FUNCTION_BLOCK CROSSCOMM_PEER_870DEA938BB7E735 (* Service Interface Function Block Type *)
  (* Standard: 61499-2 *)
  (* Version 0.0, 9/22/2017, bababen, nxtControl GmbH, template *)
  PACKAGE Main;
  (* Compiler Cpp nxtControl builtin 1.0 *)
  {SET_ATTRIBUTE(Runtime.FBType.ImplementingType, Runtime.System#DYNGEN_CROSSCOMM_PEER)}
  {SET_ATTRIBUTE(Configuration.GenericFBType.InterfaceParams, Runtime.System#<InterfaceList> <EventOutputs> <Event Name="INITO"> <With Var="ExtendPusher" /> </Event> <Event Name="CNF"> <With Var="ExtendPusher" /> </Event> </EventOutputs> <OutputVars> <VarDeclaration Name="ExtendPusher" Type="BOOL" /> </OutputVars> </InterfaceList>)}
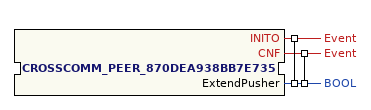
  EVENT_OUTPUT
    INITO WITH ExtendPusher;
    CNF WITH ExtendPusher;
  END_EVENT
  VAR_OUTPUT
    ExtendPusher : BOOL;
  END_VAR
  EC_STATES
    START;
  END_STATES
END_FUNCTION_BLOCK
